Fanuc TP program (LS listing): dropconv4.ls

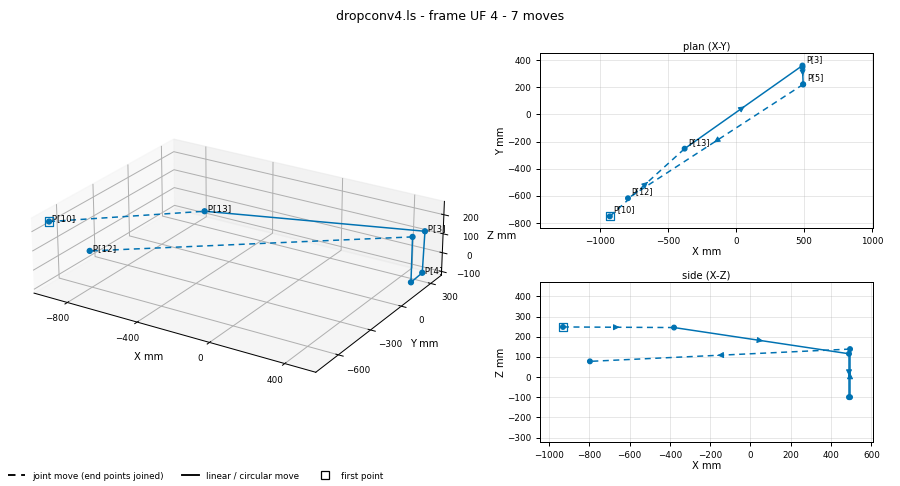
[picture p0: tool path of dropconv4.ls in frame UF 4, 7 of 7 moves have a stored position in this frame; points joined in program order, loops and branches not executed]
/PROG  DROPCONV4
/ATTR
OWNER		= MNEDITOR;
COMMENT		= "";
PROG_SIZE	= 1205;
CREATE		= DATE 26-02-24  TIME 08:56:10;
MODIFIED	= DATE 26-02-24  TIME 08:56:10;
FILE_NAME	= DROPCONV;
VERSION		= 0;
LINE_COUNT	= 29;
MEMORY_SIZE	= 1477;
PROTECT		= READ_WRITE;
TCD:  STACK_SIZE	= 0,
      TASK_PRIORITY	= 50,
      TIME_SLICE	= 0,
      BUSY_LAMP_OFF	= 0,
      ABORT_REQUEST	= 0,
      PAUSE_REQUEST	= 0;
DEFAULT_GROUP	= 1,*,*,*,*;
CONTROL_CODE	= 00000000 00000000;
LOCAL_REGISTERS	= 0,0,0;
/APPL
/MN
   1:  !***************** ;
   2:  !Drop de pieza ;
   3:  !Banda 2 de Conveyor ;
   4:  !***************** ;
   5:   ;
   6:  UTOOL_NUM=1 ;
   7:  UFRAME_NUM=4 ;
   8:  PAYLOAD[2] ;
   9:  TIMER[5]=RESET ;
  10:  TIMER[5]=START ;
  11:   ;
  12:J P[10] 100% CNT80    ;
  13:   ;
  14:J P[13] 100% CNT100    ;
  15:L P[3] 1000mm/sec CNT10    ;
  16:L P[4] 500mm/sec FINE    ;
  17:   ;
  18:  CALL CIL1_EXTENDER    ;
  19:   ;
  20:L P[5] 800mm/sec CNT10    ;
  21:  DO[19:OFF:(Reserved)]=PULSE,1.0sec ;
  22:L P[6] 1500mm/sec CNT30    ;
  23:J P[12] 100% CNT100    ;
  24:   ;
  25:  CALL CIL2_EXTENDER    ;
  26:  R[101:Proceso]=0    ;
  27:  R[198]=0    ;
  28:  F[2:OFF:(Reserved)]=(OFF) ;
  29:  TIMER[5]=STOP ;
/POS
P[3]{
   GP1:
	UF : 4, UT : 1,		CONFIG : 'N U T, 0, 0, 0',
	X =   488.570  mm,	Y =   360.379  mm,	Z =   115.889  mm,
	W =  -179.643 deg,	P =    -1.154 deg,	R =    93.280 deg
};
P[4]{
   GP1:
	UF : 4, UT : 1,		CONFIG : 'N U T, 0, 0, 0',
	X =   488.570  mm,	Y =   348.023  mm,	Z =   -99.396  mm,
	W =  -179.643 deg,	P =    -1.154 deg,	R =    93.280 deg
};
P[5]{
   GP1:
	UF : 4, UT : 1,		CONFIG : 'N U T, 0, 0, 0',
	X =   493.710  mm,	Y =   221.681  mm,	Z =   -99.396  mm,
	W =  -179.643 deg,	P =    -1.154 deg,	R =    93.280 deg
};
P[6]{
   GP1:
	UF : 4, UT : 1,		CONFIG : 'N U T, 0, 0, 0',
	X =   493.710  mm,	Y =   221.681  mm,	Z =   139.175  mm,
	W =  -179.643 deg,	P =    -1.154 deg,	R =    93.280 deg
};
P[10]{
   GP1:
	UF : 4, UT : 1,		CONFIG : 'N U T, 0, 0, 0',
	X =  -930.001  mm,	Y =  -750.257  mm,	Z =   248.875  mm,
	W =  -179.965 deg,	P =     1.349 deg,	R =   152.619 deg
};
P[12]{
   GP1:
	UF : 4, UT : 1,		CONFIG : 'N U T, 0, 0, 0',
	X =  -796.299  mm,	Y =  -616.809  mm,	Z =    78.278  mm,
	W =   179.658 deg,	P =     -.581 deg,	R =   157.820 deg
};
P[13]{
   GP1:
	UF : 4, UT : 1,		CONFIG : 'N U T, 0, 0, 0',
	X =  -379.195  mm,	Y =  -251.732  mm,	Z =   245.957  mm,
	W =   179.074 deg,	P =      .213 deg,	R =    86.372 deg
};
/END
